FUNCTION averageCalculator : REAL
VAR_INPUT
	inputbuffer : ARRAY[0..99] OF REAL;
END_VAR
VAR
	tempIndex : INT := 0;
	tempSum :REAL := 0;
END_VAR

FOR tempIndex := 0 TO 99 DO
	tempSum := tempSum + inputbuffer[tempIndex];
END_FOR
averageCalculator := tempSum/100;
RETURN;

END_FUNCTION

(* stored: Version 1.1.0.1, ProductVersion 3.1.4024.13
   POU averageCalculator: Id {b0aa6b54-c0c9-412d-b848-9ffba4329aa3}, SpecialFunc None *)
